// TIA Portal project "TestProject1" (V17)

(* hardware
DEVICE "PC-System_0"  IPC627D PN/IE
   slot 0: "PC-System_0"  IPC627D PN/IE  6AG4131-2xxxx-xxxx
      slot 124: "Diagbase"  Diagbase  V6.0.4
      slot 125: "PC-System_0"  PC Station 2.2  Station_Manager  V2.2
   slot 2: "Software PLC_0"  CPU 1507S F  6ES7 672-7FC01-0YA0  V2.1
      slot 3: "CPU display_1"  6ES7591-1BA00-0AA0
   slot 100: "PROFINET onboard_1"  PROFINET Interface  V7.1.0
      slot 1: "PROFINET Interface_1"  PROFINET Interface
         slot 1: "Port_1"  Port
   slot 101: "PROFINET onboard_2"  PROFINET Interface  V7.1.0
      slot 1: "PROFINET Interface_1"  PROFINET Interface
         slot 1: "Port_1"  Port
DEVICE "S71500/ET200MP station_1"  S7-1500 station
   slot 0: "Rail_0"  Rack  6ES7 590-1***0-0AA0
   slot 1: "PLC_0"  CPU 1511-1 PN  6ES7 511-1AK01-0AB0  V2.1
      slot 3: "CPU display_1"  6ES7591-1AA00-0AA0
DEVICE "HMI_0"  TP1500 Basic color PN
   slot 0: "TP1500 Basic color PN"  TP1500 Basic color PN  6AV6 647-0AG11-3AX0  12.0.0.0
   slot 1: "HMI_RT_1"  TP1500 Basic color PN  6AV6 647-0AG11-3AX0  12.0.0.0
   slot 5: "HMI_0.IE_CP_1"  PROFINET Interface  12.0.0.0
      slot 1: "PROFINET Interface_1"  PROFINET Interface
         slot 1: "Port_1"  Port
DEVICE "S71500/ET200MP station_2"  S7-1500 station
   slot 0: "Rail_0"  Rack  6ES7 590-1***0-0AA0
   slot 1: "PLC_1"  CPU 1511-1 PN  6ES7 511-1AK01-0AB0  V2.1
      slot 3: "CPU display_1"  6ES7591-1AA00-0AA0
DEVICE "S71500/ET200MP station_3"  S7-1500 station
   slot 0: "Rail_0"  Rack  6ES7 590-1***0-0AA0
   slot 1: "PLC_1.1"  CPU 1511-1 PN  6ES7 511-1AK01-0AB0  V2.1
      slot 3: "CPU display_1"  6ES7591-1AA00-0AA0
DEVICE "S71500/ET200MP station_4"  S7-1500 station
   slot 0: "Rail_0"  Rack  6ES7 590-1***0-0AA0
   slot 1: "PLC_1.1.1"  CPU 1511-1 PN  6ES7 511-1AK01-0AB0  V2.1
      slot 3: "CPU display_1"  6ES7591-1AA00-0AA0
DEVICE "PC-System_1"  IPC627D PN/IE
   slot 0: "PC-System_1"  IPC627D PN/IE  6AG4131-2xxxx-xxxx
      slot 124: "Diagbase"  Diagbase  V6.0.4
      slot 125: "PC-System_1"  PC Station 2.2  Station_Manager  V2.2
   slot 2: "Software PLC_1"  CPU 1507S F  6ES7 672-7FC01-0YA0  V2.1
      slot 3: "CPU display_1"  6ES7591-1BA00-0AA0
   slot 100: "PROFINET onboard_1"  PROFINET Interface  V7.1.0
      slot 1: "PROFINET Interface_1"  PROFINET Interface
         slot 1: "Port_1"  Port
   slot 101: "PROFINET onboard_2"  PROFINET Interface  V7.1.0
      slot 1: "PROFINET Interface_1"  PROFINET Interface
         slot 1: "Port_1"  Port
DEVICE "PC-System_1.1"  IPC627D PN/IE
   slot 0: "PC-System_2"  IPC627D PN/IE  6AG4131-2xxxx-xxxx
      slot 124: "Diagbase"  Diagbase  V6.0.4
      slot 125: "PC-System_2"  PC Station 2.2  Station_Manager  V2.2
   slot 2: "Software PLC_1.1"  CPU 1507S F  6ES7 672-7FC01-0YA0  V2.1
      slot 3: "CPU display_1"  6ES7591-1BA00-0AA0
   slot 100: "PROFINET onboard_1"  PROFINET Interface  V7.1.0
      slot 1: "PROFINET Interface_1"  PROFINET Interface
         slot 1: "Port_1"  Port
   slot 101: "PROFINET onboard_2"  PROFINET Interface  V7.1.0
      slot 1: "PROFINET Interface_1"  PROFINET Interface
         slot 1: "Port_1"  Port
DEVICE "PC-System_1.1.1"  IPC627D PN/IE
   slot 0: "PC-System_1.1_1"  IPC627D PN/IE  6AG4131-2xxxx-xxxx
      slot 124: "Diagbase"  Diagbase  V6.0.4
      slot 125: "PC-System_1.1_1"  PC Station 2.2  Station_Manager  V2.2
   slot 2: "Software PLC_1.1.1"  CPU 1507S F  6ES7 672-7FC01-0YA0  V2.1
      slot 3: "CPU display_1"  6ES7591-1BA00-0AA0
   slot 100: "PROFINET onboard_1"  PROFINET Interface  V7.1.0
      slot 1: "PROFINET Interface_1"  PROFINET Interface
         slot 1: "Port_1"  Port
   slot 101: "PROFINET onboard_2"  PROFINET Interface  V7.1.0
      slot 1: "PROFINET Interface_1"  PROFINET Interface
         slot 1: "Port_1"  Port
*)

// ===== PLC "Software PLC_0"  CPU 1507S F =====
// protected blocks, not shown: "Main_Safety_RTG1", "Main_Safety_RTG1_DB"

VAR_GLOBAL   // PLC tag table "Default tag table"
   "Tag_1" AT %M0.0 : Bool;
END_VAR

ORGANIZATION_BLOCK "Main"   // OB1, LAD, ProgramCycle
TITLE = "Main Program Sweep (Cycle)"
{ S7_Optimized_Access := 'TRUE' }
VERSION : 0.1
   VAR_INPUT
      Initial_Call : Bool;   // Initial call of this OB
      Remanence : Bool;   // =True, if remanent data are available
   END_VAR
BEGIN
END_ORGANIZATION_BLOCK

// folder: 0_OBs

ORGANIZATION_BLOCK "OB_CYC_IN_100ms"   // OB31, LAD, CyclicInterrupt
{ S7_Optimized_Access := 'TRUE' }
VERSION : 0.1
   VAR_INPUT
      Initial_Call : Bool;   // Initial call of this OB
      Event_Count : Int;   // Events discarded
   END_VAR
BEGIN

REGION Network 1
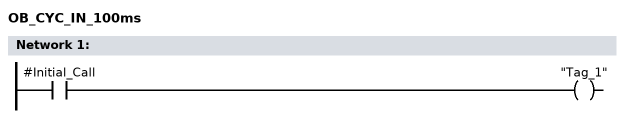
   RUNG wire#powerrail
      Contact( #Initial_Call )
      Coil( "Tag_1" )
   END_RUNG
   // the same network as SCL:
   "Tag_1" := #Initial_Call;
END_REGION
END_ORGANIZATION_BLOCK

ORGANIZATION_BLOCK "Startup"   // OB100, LAD, Startup
TITLE = "Complete Restart"
{ S7_Optimized_Access := 'TRUE' }
VERSION : 0.1
   VAR_INPUT
      LostRetentive : Bool;   // True if retentive data are lost
      LostRTC : Bool;   // True if date and time are lost
   END_VAR
BEGIN
END_ORGANIZATION_BLOCK

ORGANIZATION_BLOCK "Programming error"   // OB121, LAD, ProgrammingError
{ S7_Optimized_Access := 'TRUE' }
VERSION : 0.1
   VAR_INPUT
      BlockNr : UInt;   // Number of causing block
      Reaction : USInt;   // 0:ignore, 1:substitute, 2:skip
      Fault_ID : Byte;   // Fault identifier
      BlockType : USInt;   // 16#01:OB, 16#02:FC, 16#03:FB, 16#04:SFC, 16#05:SFB, 16#06:DB: Type of block causing the error
      Area : USInt;   // Area where the error occured
      DBNr : DB_ANY;   // DB number if Area = DB or DI
      Csg_OBNr : OB_Any;   // Number of OB causing the error
      Csg_Prio : USInt;   // Priority of OB causing the error
      Width : USInt;   // 0:bit, 1:byte, 2:word, 3:dword, 4:lword
   END_VAR
BEGIN
END_ORGANIZATION_BLOCK

ORGANIZATION_BLOCK "Main_1"   // OB123, LAD, ProgramCycle
TITLE = "Main Program Sweep (Cycle)"
{ S7_Optimized_Access := 'TRUE' }
VERSION : 0.1
   VAR_INPUT
      Initial_Call : Bool;   // Initial call of this OB
      Remanence : Bool;   // =True, if remanent data are available
   END_VAR
BEGIN
END_ORGANIZATION_BLOCK

// ===== PLC "PLC_0"  CPU 1511-1 PN =====

VAR_GLOBAL   // PLC tag table "Default tag table"
   "Tag_1" AT %M0.0 : Bool;
   "Tag_2" AT %M0.1 : Bool;
   "Tag_3" AT %M0.2 : Bool;
   "Tag_4" AT %M1.0 : Bool;
   "Tag_5" AT %M1.1 : Bool;
   "Tag_6" AT %M0.4 : Bool;
   "Tag_7" AT %M0.5 : Bool;
END_VAR

// folder: Common/CarrierRegister

TYPE "ML_SubstratState"
   STRUCT
      Present : Bool;
      Good : Bool;
      PM1_1_Sputtered : Bool;
      PM1_2_Sputtered : Bool;
      PM1_3_Sputtered : Bool;
      PM1_x_Sputtered : Bool;
      PM2_1_Sputtered : Bool;
      PM2_2_Sputtered : Bool;
      PM2_3_Sputtered : Bool;
      PM2_x_Sputtered : Bool;
      PM3_1_Sputtered : Bool;
      PM3_2_Sputtered : Bool;
      PM3_3_Sputtered : Bool;
      PM3_x_Sputtered : Bool;
   END_STRUCT;
END_TYPE

TYPE "ML_SubstratInformation"
   STRUCT
      P_Substrate : Struct
         Offset : DInt;
         State : Byte;
         ProcessState : "ML_SubstratState";
         MeasuringFlags : Byte;
         ConveyingThroughFlags : Byte;
         ID : String[15];
         CoverCounter : Byte;
         ColorFlags : Byte;
      END_STRUCT;
   END_STRUCT;
END_TYPE

TYPE "ML_ChamberSubstrateRegister"
   STRUCT
      LM1 : "ML_CarrierRegisterShort";
      LL1 : "ML_CarrierRegisterShort";
      EC1 : "ML_CarrierRegisterShort";
      PM1 : "ML_CarrierRegisterShort";
      EC2 : "ML_CarrierRegisterShort";
   END_STRUCT;
END_TYPE

TYPE "ML_CarrierRegisterShort"
   STRUCT
      ID : Int;
      ArrayIndex : Int;
      ColorFlags : Byte;
      CoverCounter : Int;
      Content : Struct
         Substrate_1 : "ML_SubstratInformation";
         Substrate_2 : "ML_SubstratInformation";
      END_STRUCT;
   END_STRUCT;
END_TYPE

// folder: 1_Tests

DATA_BLOCK "DB_block_1"   // DB1
{ S7_Optimized_Access := 'TRUE' }
VERSION : 0.1
   VAR
      Header : ArrayDBHeader;
      THIS : Array[0..100] of Bool;
   END_VAR
BEGIN
   Header.LowerBound := 0;
   Header.UpperBound := 100;
   Header.Elements := 101;
   Header.PaddedSize := 1;
   Header.ElementSize := 1;
END_DATA_BLOCK

// folder: Common/CarrierRegister

DATA_BLOCK "GLOBAL_POSITIONING"   // DB54
{ S7_Optimized_Access := 'TRUE' }
VERSION : 0.1
   VAR
      SubstratRegister : "ML_ChamberSubstrateRegister";
   END_VAR
BEGIN
END_DATA_BLOCK

// folder: 0_OBs

ORGANIZATION_BLOCK "OB_CYC_IN_100ms"   // OB31, LAD, CyclicInterrupt
{ S7_Optimized_Access := 'TRUE' }
VERSION : 0.1
   VAR_INPUT
      Initial_Call : Bool;   // Initial call of this OB
      Event_Count : Int;   // Events discarded
   END_VAR
BEGIN

REGION Network 1
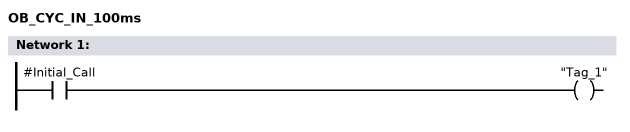
   RUNG wire#powerrail
      Contact( #Initial_Call )
      Coil( "Tag_1" )
   END_RUNG
   // the same network as SCL:
   "Tag_1" := #Initial_Call;
END_REGION
END_ORGANIZATION_BLOCK

ORGANIZATION_BLOCK "Startup"   // OB100, LAD, Startup
TITLE = "Complete Restart"
{ S7_Optimized_Access := 'TRUE' }
VERSION : 0.1
   VAR_INPUT
      LostRetentive : Bool;   // True if retentive data are lost
      LostRTC : Bool;   // True if date and time are lost
   END_VAR
BEGIN
END_ORGANIZATION_BLOCK

ORGANIZATION_BLOCK "Programming error"   // OB121, LAD, ProgrammingError
{ S7_Optimized_Access := 'TRUE' }
VERSION : 0.1
   VAR_INPUT
      BlockNr : UInt;   // Number of causing block
      Reaction : USInt;   // 0:ignore, 1:substitute, 2:skip
      Fault_ID : Byte;   // Fault identifier
      BlockType : USInt;   // 16#01:OB, 16#02:FC, 16#03:FB, 16#04:SFC, 16#05:SFB, 16#06:DB: Type of block causing the error
      Area : USInt;   // Area where the error occured
      DBNr : DB_ANY;   // DB number if Area = DB or DI
      Csg_OBNr : OB_Any;   // Number of OB causing the error
      Csg_Prio : USInt;   // Priority of OB causing the error
      Width : USInt;   // 0:bit, 1:byte, 2:word, 3:dword, 4:lword
   END_VAR
BEGIN
END_ORGANIZATION_BLOCK

ORGANIZATION_BLOCK "Main_1"   // OB123, LAD, ProgramCycle
TITLE = "Main Program Sweep (Cycle)"
{ S7_Optimized_Access := 'TRUE' }
VERSION : 0.1
   VAR_INPUT
      Initial_Call : Bool;   // Initial call of this OB
      Remanence : Bool;   // =True, if remanent data are available
   END_VAR
BEGIN

REGION Network 1
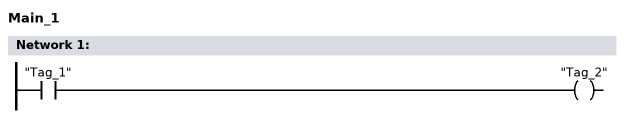
   RUNG wire#powerrail
      Contact( "Tag_1" )
      Coil( "Tag_2" )
   END_RUNG
   // the same network as SCL:
   "Tag_2" := "Tag_1";
END_REGION
END_ORGANIZATION_BLOCK

// folder: 1_Tests

FUNCTION "FC_Block_1" : Void   // FC1, SCL
{ S7_Optimized_Access := 'TRUE' }
VERSION : 0.1
BEGIN
   IF "Tag_6" THEN
       // Statement section IF
       "Tag_2" := FALSE;
   END_IF;
END_FUNCTION

// ===== PLC "PLC_1"  CPU 1511-1 PN =====

VAR_GLOBAL   // PLC tag table "Default tag table"
   "Tag_1" AT %M0.0 : Bool;
END_VAR

// folder: Data

DATA_BLOCK "DataBlock1"   // DB1
{ S7_Optimized_Access := 'TRUE' }
VERSION : 0.1
BEGIN
END_DATA_BLOCK

// folder: 0_OBs

ORGANIZATION_BLOCK "OB_CYC_IN_100ms"   // OB31, LAD, CyclicInterrupt
{ S7_Optimized_Access := 'TRUE' }
VERSION : 0.1
   VAR_INPUT
      Initial_Call : Bool;   // Initial call of this OB
      Event_Count : Int;   // Events discarded
   END_VAR
BEGIN

REGION Network 1
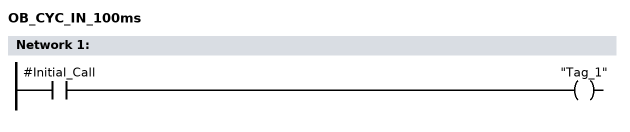
   RUNG wire#powerrail
      Contact( #Initial_Call )
      Coil( "Tag_1" )
   END_RUNG
   // the same network as SCL:
   "Tag_1" := #Initial_Call;
END_REGION
END_ORGANIZATION_BLOCK

ORGANIZATION_BLOCK "Startup"   // OB100, LAD, Startup
TITLE = "Complete Restart"
{ S7_Optimized_Access := 'TRUE' }
VERSION : 0.1
   VAR_INPUT
      LostRetentive : Bool;   // True if retentive data are lost
      LostRTC : Bool;   // True if date and time are lost
   END_VAR
BEGIN
END_ORGANIZATION_BLOCK

ORGANIZATION_BLOCK "Programming error"   // OB121, LAD, ProgrammingError
{ S7_Optimized_Access := 'TRUE' }
VERSION : 0.1
   VAR_INPUT
      BlockNr : UInt;   // Number of causing block
      Reaction : USInt;   // 0:ignore, 1:substitute, 2:skip
      Fault_ID : Byte;   // Fault identifier
      BlockType : USInt;   // 16#01:OB, 16#02:FC, 16#03:FB, 16#04:SFC, 16#05:SFB, 16#06:DB: Type of block causing the error
      Area : USInt;   // Area where the error occured
      DBNr : DB_ANY;   // DB number if Area = DB or DI
      Csg_OBNr : OB_Any;   // Number of OB causing the error
      Csg_Prio : USInt;   // Priority of OB causing the error
      Width : USInt;   // 0:bit, 1:byte, 2:word, 3:dword, 4:lword
   END_VAR
BEGIN
END_ORGANIZATION_BLOCK

ORGANIZATION_BLOCK "Main_1"   // OB123, LAD, ProgramCycle
TITLE = "Main Program Sweep (Cycle)"
{ S7_Optimized_Access := 'TRUE' }
VERSION : 0.1
   VAR_INPUT
      Initial_Call : Bool;   // Initial call of this OB
      Remanence : Bool;   // =True, if remanent data are available
   END_VAR
BEGIN
END_ORGANIZATION_BLOCK

// folder: Code

FUNCTION "FC_Function1" : Void   // FC1, SCL
{ S7_Optimized_Access := 'TRUE' }
VERSION : 0.1
BEGIN
END_FUNCTION

// ===== PLC "PLC_1.1"  CPU 1511-1 PN =====

VAR_GLOBAL   // PLC tag table "Default tag table"
   "Tag_1" AT %M0.0 : Bool;
END_VAR

ORGANIZATION_BLOCK "Main"   // OB1, LAD, ProgramCycle
TITLE = "Main Program Sweep (Cycle)"
{ S7_Optimized_Access := 'TRUE' }
VERSION : 0.1
   VAR_INPUT
      Initial_Call : Bool;   // Initial call of this OB
      Remanence : Bool;   // =True, if remanent data are available
   END_VAR
BEGIN
END_ORGANIZATION_BLOCK

// folder: 0_OBs

ORGANIZATION_BLOCK "OB_CYC_IN_100ms"   // OB31, LAD, CyclicInterrupt
{ S7_Optimized_Access := 'TRUE' }
VERSION : 0.1
   VAR_INPUT
      Initial_Call : Bool;   // Initial call of this OB
      Event_Count : Int;   // Events discarded
   END_VAR
BEGIN

REGION Network 1
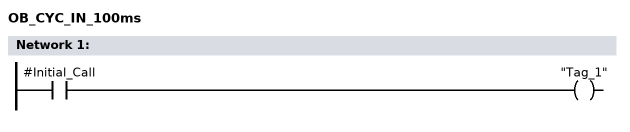
   RUNG wire#powerrail
      Contact( #Initial_Call )
      Coil( "Tag_1" )
   END_RUNG
   // the same network as SCL:
   "Tag_1" := #Initial_Call;
END_REGION
END_ORGANIZATION_BLOCK

ORGANIZATION_BLOCK "Startup"   // OB100, LAD, Startup
TITLE = "Complete Restart"
{ S7_Optimized_Access := 'TRUE' }
VERSION : 0.1
   VAR_INPUT
      LostRetentive : Bool;   // True if retentive data are lost
      LostRTC : Bool;   // True if date and time are lost
   END_VAR
BEGIN
END_ORGANIZATION_BLOCK

ORGANIZATION_BLOCK "Programming error"   // OB121, LAD, ProgrammingError
{ S7_Optimized_Access := 'TRUE' }
VERSION : 0.1
   VAR_INPUT
      BlockNr : UInt;   // Number of causing block
      Reaction : USInt;   // 0:ignore, 1:substitute, 2:skip
      Fault_ID : Byte;   // Fault identifier
      BlockType : USInt;   // 16#01:OB, 16#02:FC, 16#03:FB, 16#04:SFC, 16#05:SFB, 16#06:DB: Type of block causing the error
      Area : USInt;   // Area where the error occured
      DBNr : DB_ANY;   // DB number if Area = DB or DI
      Csg_OBNr : OB_Any;   // Number of OB causing the error
      Csg_Prio : USInt;   // Priority of OB causing the error
      Width : USInt;   // 0:bit, 1:byte, 2:word, 3:dword, 4:lword
   END_VAR
BEGIN
END_ORGANIZATION_BLOCK

ORGANIZATION_BLOCK "Main_1"   // OB123, LAD, ProgramCycle
TITLE = "Main Program Sweep (Cycle)"
{ S7_Optimized_Access := 'TRUE' }
VERSION : 0.1
   VAR_INPUT
      Initial_Call : Bool;   // Initial call of this OB
      Remanence : Bool;   // =True, if remanent data are available
   END_VAR
BEGIN
END_ORGANIZATION_BLOCK

// ===== PLC "PLC_1.1.1"  CPU 1511-1 PN =====

VAR_GLOBAL   // PLC tag table "Default tag table"
   "Tag_1" AT %M0.0 : Bool;
END_VAR

ORGANIZATION_BLOCK "Main"   // OB1, LAD, ProgramCycle
TITLE = "Main Program Sweep (Cycle)"
{ S7_Optimized_Access := 'TRUE' }
VERSION : 0.1
   VAR_INPUT
      Initial_Call : Bool;   // Initial call of this OB
      Remanence : Bool;   // =True, if remanent data are available
   END_VAR
BEGIN
END_ORGANIZATION_BLOCK

// ===== PLC "Software PLC_1"  CPU 1507S F =====
// protected blocks, not shown: "Main_Safety_RTG1", "Main_Safety_RTG1_DB"

VAR_GLOBAL   // PLC tag table "Default tag table"
   "Tag_1" AT %M0.0 : Bool;
END_VAR

ORGANIZATION_BLOCK "Main"   // OB1, LAD, ProgramCycle
TITLE = "Main Program Sweep (Cycle)"
{ S7_Optimized_Access := 'TRUE' }
VERSION : 0.1
   VAR_INPUT
      Initial_Call : Bool;   // Initial call of this OB
      Remanence : Bool;   // =True, if remanent data are available
   END_VAR
BEGIN
END_ORGANIZATION_BLOCK

// folder: 0_OBs

ORGANIZATION_BLOCK "OB_CYC_IN_100ms"   // OB31, LAD, CyclicInterrupt
{ S7_Optimized_Access := 'TRUE' }
VERSION : 0.1
   VAR_INPUT
      Initial_Call : Bool;   // Initial call of this OB
      Event_Count : Int;   // Events discarded
   END_VAR
BEGIN

REGION Network 1
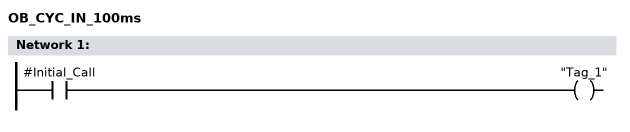
   RUNG wire#powerrail
      Contact( #Initial_Call )
      Coil( "Tag_1" )
   END_RUNG
   // the same network as SCL:
   "Tag_1" := #Initial_Call;
END_REGION
END_ORGANIZATION_BLOCK

ORGANIZATION_BLOCK "Startup"   // OB100, LAD, Startup
TITLE = "Complete Restart"
{ S7_Optimized_Access := 'TRUE' }
VERSION : 0.1
   VAR_INPUT
      LostRetentive : Bool;   // True if retentive data are lost
      LostRTC : Bool;   // True if date and time are lost
   END_VAR
BEGIN
END_ORGANIZATION_BLOCK

ORGANIZATION_BLOCK "Programming error"   // OB121, LAD, ProgrammingError
{ S7_Optimized_Access := 'TRUE' }
VERSION : 0.1
   VAR_INPUT
      BlockNr : UInt;   // Number of causing block
      Reaction : USInt;   // 0:ignore, 1:substitute, 2:skip
      Fault_ID : Byte;   // Fault identifier
      BlockType : USInt;   // 16#01:OB, 16#02:FC, 16#03:FB, 16#04:SFC, 16#05:SFB, 16#06:DB: Type of block causing the error
      Area : USInt;   // Area where the error occured
      DBNr : DB_ANY;   // DB number if Area = DB or DI
      Csg_OBNr : OB_Any;   // Number of OB causing the error
      Csg_Prio : USInt;   // Priority of OB causing the error
      Width : USInt;   // 0:bit, 1:byte, 2:word, 3:dword, 4:lword
   END_VAR
BEGIN
END_ORGANIZATION_BLOCK

ORGANIZATION_BLOCK "Main_1"   // OB123, LAD, ProgramCycle
TITLE = "Main Program Sweep (Cycle)"
{ S7_Optimized_Access := 'TRUE' }
VERSION : 0.1
   VAR_INPUT
      Initial_Call : Bool;   // Initial call of this OB
      Remanence : Bool;   // =True, if remanent data are available
   END_VAR
BEGIN
END_ORGANIZATION_BLOCK

// ===== PLC "Software PLC_1.1"  CPU 1507S F =====
// protected blocks, not shown: "Main_Safety_RTG1", "Main_Safety_RTG1_DB"

VAR_GLOBAL   // PLC tag table "Default tag table"
   "Tag_1" AT %M0.0 : Bool;
END_VAR

ORGANIZATION_BLOCK "Main"   // OB1, LAD, ProgramCycle
TITLE = "Main Program Sweep (Cycle)"
{ S7_Optimized_Access := 'TRUE' }
VERSION : 0.1
   VAR_INPUT
      Initial_Call : Bool;   // Initial call of this OB
      Remanence : Bool;   // =True, if remanent data are available
   END_VAR
BEGIN
END_ORGANIZATION_BLOCK

// folder: 0_OBs

ORGANIZATION_BLOCK "OB_CYC_IN_100ms"   // OB31, LAD, CyclicInterrupt
{ S7_Optimized_Access := 'TRUE' }
VERSION : 0.1
   VAR_INPUT
      Initial_Call : Bool;   // Initial call of this OB
      Event_Count : Int;   // Events discarded
   END_VAR
BEGIN

REGION Network 1
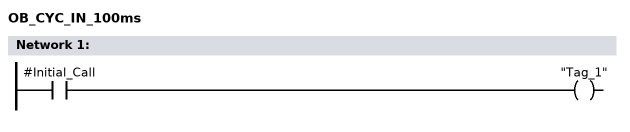
   RUNG wire#powerrail
      Contact( #Initial_Call )
      Coil( "Tag_1" )
   END_RUNG
   // the same network as SCL:
   "Tag_1" := #Initial_Call;
END_REGION
END_ORGANIZATION_BLOCK

ORGANIZATION_BLOCK "Startup"   // OB100, LAD, Startup
TITLE = "Complete Restart"
{ S7_Optimized_Access := 'TRUE' }
VERSION : 0.1
   VAR_INPUT
      LostRetentive : Bool;   // True if retentive data are lost
      LostRTC : Bool;   // True if date and time are lost
   END_VAR
BEGIN
END_ORGANIZATION_BLOCK

ORGANIZATION_BLOCK "Programming error"   // OB121, LAD, ProgrammingError
{ S7_Optimized_Access := 'TRUE' }
VERSION : 0.1
   VAR_INPUT
      BlockNr : UInt;   // Number of causing block
      Reaction : USInt;   // 0:ignore, 1:substitute, 2:skip
      Fault_ID : Byte;   // Fault identifier
      BlockType : USInt;   // 16#01:OB, 16#02:FC, 16#03:FB, 16#04:SFC, 16#05:SFB, 16#06:DB: Type of block causing the error
      Area : USInt;   // Area where the error occured
      DBNr : DB_ANY;   // DB number if Area = DB or DI
      Csg_OBNr : OB_Any;   // Number of OB causing the error
      Csg_Prio : USInt;   // Priority of OB causing the error
      Width : USInt;   // 0:bit, 1:byte, 2:word, 3:dword, 4:lword
   END_VAR
BEGIN
END_ORGANIZATION_BLOCK

ORGANIZATION_BLOCK "Main_1"   // OB123, LAD, ProgramCycle
TITLE = "Main Program Sweep (Cycle)"
{ S7_Optimized_Access := 'TRUE' }
VERSION : 0.1
   VAR_INPUT
      Initial_Call : Bool;   // Initial call of this OB
      Remanence : Bool;   // =True, if remanent data are available
   END_VAR
BEGIN
END_ORGANIZATION_BLOCK

// ===== PLC "Software PLC_1.1.1"  CPU 1507S F =====
// protected blocks, not shown: "Main_Safety_RTG1", "Main_Safety_RTG1_DB"

ORGANIZATION_BLOCK "Main"   // OB1, LAD, ProgramCycle
TITLE = "Main Program Sweep (Cycle)"
{ S7_Optimized_Access := 'TRUE' }
VERSION : 0.1
   VAR_INPUT
      Initial_Call : Bool;   // Initial call of this OB
      Remanence : Bool;   // =True, if remanent data are available
   END_VAR
BEGIN
END_ORGANIZATION_BLOCK

(* ===== HMI "HMI_RT_1" =====
system functions are stored by id; their names below are inferred from use

HMI tags "Default tag table"
   "Tag_ScreenNumber" : UInt, internal

Template "Template_1" 1024x768
   Button "Exit" at 943,707 size 79x59; TextOff 'Exit'; PictureOff "ExitRuntime_TP1500_Basic_color_PN"; PictureOn "ExitRuntime_TP1500_Basic_color_PN"
      on Release: StopRuntime(0)
   Button "Template_Button" at 857,707 size 79x59; TextOff 'Text'
   Button "Template_Button_1" at 772,707 size 79x59; TextOff 'Text'
   Button "Template_Button_2" at 686,707 size 79x59; TextOff 'Text'
   Button "Template_Button_3" at 600,707 size 79x59; TextOff 'Text'
   Button "Template_Button_4" at 515,707 size 79x59; TextOff 'Text'
   Button "Template_Button_5" at 429,707 size 79x59; TextOff 'Text'
   Button "Template_Button_6" at 344,707 size 79x59; TextOff 'Text'
   Button "Template_Button_7" at 258,707 size 79x59; TextOff 'Text'
   Button "Template_Button_8" at 172,707 size 79x59; TextOff 'Text'
   Button "Template_Button_9" at 87,707 size 79x59; TextOff 'Text'
   Button "Start screen" at 1,707 size 79x59; TextOff 'Start screen'; PictureOff "NavigateHome_TP1500_Basic_color_PN"; PictureOn "NavigateHome_TP1500_Basic_color_PN"
      on Release: ActivateScreen("Root screen", 0)
   SymbolicIOField "Symbolic_IO_Field_Screen" at 109,11 size 808x35; TextOff '0'; TextOn '1'; TextList "TextList_ScreenNames"
      ProcessValue <- "Tag_ScreenNumber"
      on Change: ActivateScreenByNumber("Tag_ScreenNumber", 0)
   DateTimeField "HmiScreenItemData" at 919,30 size 105x30
   DateTimeField "HmiScreenItemData_1" at 919,0 size 105x30
   GraphicView "Logo" at 0,0 size 107x60; Picture "Logo of HMI_0"

screen "Root screen" 1024x768, template "Template_1"
   on GenerateScreen: SetTag("Tag_ScreenNumber", 1)
   TextField "HmiScreenItemData" at 103,370 size 819x23; Text 'Welcome to HMI_0 (TP1500 Basic color PN)!'
*)